// TIA Portal V17 export
// export: Created 2025-06-25T13:13:32.2183109Z, ExportSetting WithDefaults, DisplayName Totally Integrated Automation Portal, DisplayVersion V17 Update 8, DisplayName TIA Portal Openness, DisplayVersion V17 Update 8, DisplayName TIA Portal Version Control Interface, DisplayVersion V17, DisplayName STEP 7 Professional, DisplayVersion V17 Update 8, DisplayName STEP 7 Safety, DisplayVersion V17 Update 6, DisplayName WinCC Advanced, DisplayVersion V17 Update 8
TYPE "PerformanceControl-STRUCT"
// stored: IsFailsafeCompliant false
   STRUCT
      MinimumPerformanceRate : Real := 0.0;   // [%]
      SwitchToStandby_timeDelay : Time := T#0s;   // Switches off the engine if the required performance value unterruns minimum perofrmance value for this time. Deactivated if zero
      HeatSink : Struct
         Control_Active : Bool := true;   // 1 = enable controller, 0 = disable controller
         UseFeedFlow : Bool := true;   // 1 = use feed flow, 0 = use return flow
         Setpoint : Real;
         DT_Limit_Standby : Real := 20.0;   // Go to standby
         DT_Limit_Resume : Real := 0.5;   // Resume operation
         Kp : Real := 10.0;   // Proportional gain
         Tn : Real := 60.0;   // Integral gain (reset time)
      END_STRUCT;
      HeatSource : Struct
         Control_Active : Bool := true;   // 1 = enable controller, 0 = disable controller
         UseFeedFlow : Bool := true;   // 1 = use feed flow, 0 = use return flow
         Setpoint : Real;
         DT_Limit_Standby : Real := 40.0;   // Go to standby
         DT_Limit_Resume : Real := 0.5;   // Resume operation
         Kp : Real := 1.0;   // Proportional gain
         Tn : Real := 30.0;   // Integral gain (reset time)
      END_STRUCT;
      VariableControl : Struct
         Control_Active : Bool := true;   // 1 = enable controller, 0 = disable controller
         ReferenceID : USInt := 0;
         Setpoint : Real;
         DT_Limit_Standby : Real := 20.0;   // Go to standby
         DT_Limit_Resume : Real := 10.0;   // Resume operation
         Kp : Real := 1.0;   // Proportional gain
         Tn : Real := 30.0;   // Integral gain (reset time)
      END_STRUCT;
      Config : Struct
         MinimumPerformanceRequirement { S7_SetPoint := 'True'} : Real;   // [%] Below this, additional superheat is required
         MaximumAdditionalSuperheat : Real;   // [C] Superheat to add at MinimumPerformanceRequirement
         INCREASEWITHNORESTRICTION : Real;   // [%/s] Default integrator gain
      END_STRUCT;
   END_STRUCT;
END_TYPE
